{attribute 'qualified_only'}
{attribute 'strict'}
{attribute 'to_string'}
TYPE E_MoveMode  :
(
    DISCRETE:=0,
    CONTINUOUS:=1,
    SYNCHRONOUS:=2,
    HOMING:=3
);
END_TYPE

(* stored: Version 1.1.0.1
   DUT E_MoveMode: Id {84e949ba-0c00-4cd0-8823-2572cfa98b29} *)
